# EPICS substitutions: db/Beckhoff_2XXX/ecmcMS2204-0002.substitutions
file "ecmc_analogInputFloat-chX.template"
{
  pattern {CH_ID, KEY, sourceName,  suffix,         EGU, PREC}
          {01,    CH,  EFU_current, "-EFUCurrent",  "A", 4   }
          {01,    CH,  PWI_voltage, "-PWIVoltage",  "V", 4   }
          {01,    CH,  PWI_current, "-PWICurrent",  "A", 4   }
}

file "ecmc_binaryInput-chX.template"
{
  pattern {CH_ID, KEY, sourceName,  suffix,       ZNAM,              ONAM          }
          {01,    CH,  PWI_warning, "-PWIAlrm",   "No PWI Warning",  "PWI Warning" }
          {01,    CH,  EFU_warning, "-EFUAlrm",   "No EFU Warning",  "EFU Warning" }
          {01,    CH,  EFU_error,   "-EFUErr",    "No EFU Error",    "EFU Error"   }
          {01,    CH,  EFU_tripped, "-EFUTrpd",   "EFU Not Tripped", "EFU Tripped" }
          {01,    CH,  EFU_enabled, "-EFUEnabld", "EFU Not Enabled", "EFU Enabled" }
}

file "ecmc_binaryOutput-chX.template"
{
  pattern {CH_ID, KEY, sourceName,  suffix       }
          {01,    CH,  EFU_enable,  "-EFUEnable" }
          {01,    CH,  EFU_control, "-EFUControl"}
          {01,    CH,  EFU_reset,   "-EFUReset"  }
}
